FUNCTION_BLOCK FB_MotionInterlocksCommon IMPLEMENTS I_MotionInterlocksCommon
VAR
    {attribute 'hide'}
    iMotionLogger 		: I_MotionLogger;
    {attribute 'hide'}
    bPowerEnabled: BOOL:=FALSE;
   // NC STO Input: TRUE if ok to move
    {attribute 'pytmc' := '
        pv: PLC:bHardwareEnable
        io: i
        field: ZNAM FALSE
        field: ONAM TRUE
        field: DESC TRUE if STO not hit
    '}
    bHardwareEnable AT %I*: BOOL ;

    // Used by the IOC to disable an axis
    {attribute 'pytmc' := '
        pv: PLC:bUserEnable
        io: io
        field: ZNAM DISABLE
        field: ONAM ENABLE
        field: DESC Used to disable power entirely for an axis
    '}
    bUserEnable: BOOL := TRUE;

    {attribute 'hide'}
    bEnable: BOOL;
    {attribute 'hide'}
    bReset : BOOL;
    {attribute 'hide'}
    sMessage : STRING;
    {attribute 'hide'}
    bError : BOOL;
    {attribute 'hide'}
    nErrorID : UDINT;
    {attribute 'hide'}
    bMoveOk : BOOL;
END_VAR

IF ( iMotionLogger = 0) THEN
    // throw an exception
    RETURN;
END_IF

bPowerEnabled := bEnable AND bHardwareEnable;
bPowerEnabled R= NOT bUserEnable;

(*test additional pre-move conditions here*)
bMoveOk := bUserEnable AND bHardwareEnable;

IF NOT bUserEnable OR NOT bHardwareEnable THEN
    bError := TRUE;
    nErrorID:= 11;
    bMoveOk := FALSE;
    IF NOT bUserEnable THEN
        sMessage := 'User enable interlock triggered!';
    ELSE
        sMessage := 'Hardware enbale interlocks triggered!';
    END_IF
END_IF

METHOD PUBLIC CallAfterInit
VAR_INPUT
    iMotionLogger : I_MotionLogger;
END_VAR
THIS^.iMotionLogger := iMotionLogger;
END_METHOD

METHOD DriveCommands
VAR_INPUT
    Enable: BOOL;
    NewMoveReq : BOOL;
END_VAR
THIS^.bEnable := Enable;
THIS^.bPowerEnabled := bEnable AND bHardwareEnable;
END_METHOD

{attribute 'monitoring' := 'variable'}
PROPERTY Error : BOOL
GET
Error := bError;
END_GET
END_PROPERTY

PROPERTY ErrorID : UDINT
GET
ErrorID := nErrorID;
END_GET
END_PROPERTY

//FB_Init is always available implicitly and it is used primarily for initialization.
//The return value is not evaluated. For a specific influence, you can also declare the
//methods explicitly and provide additional code there with the standard initialization
//code. You can evaluate the return value.
METHOD FB_Init: BOOL
VAR_INPUT
    bInitRetains: BOOL; // TRUE: the retain variables are initialized (reset warm / reset cold)
    bInCopyCode: BOOL;  // TRUE: the instance will be copied to the copy code afterward (online change)

    iMotionLogger 		: I_MotionLogger;
END_VAR
THIS^.iMotionLogger := iMotionLogger;
END_METHOD

PROPERTY HardwareEnable : BOOL
GET
END_GET
SET
bHardwareEnable := HardwareEnable;
END_SET
END_PROPERTY

PROPERTY Message : T_MAXSTRING
GET
Message := sMessage;
END_GET
END_PROPERTY

{attribute 'monitoring' := 'variable'}
PROPERTY MoveOk : BOOL
GET
MoveOk := bMoveOk;
END_GET
END_PROPERTY

{attribute 'monitoring' := 'variable'}
PROPERTY PowerEnabled : BOOL
GET
PowerEnabled :=bPowerEnabled;
END_GET
END_PROPERTY

METHOD Reset
THIS^.bError := FALSE;
THIS^.nErrorID:= 0;
THIS^.sMessage:='';
END_METHOD

PROPERTY UserEnable : BOOL
SET
bUserEnable := UserEnable;
END_SET
END_PROPERTY

END_FUNCTION_BLOCK

(* stored: Version 1.1.0.1
   POU FB_MotionInterlocksCommon: Id {b69073ed-2a55-41fc-84a9-b8fe79332e5e}, SpecialFunc None
   Method CallAfterInit: Id {bb25ce30-2def-4497-bead-4e7295fc730f}
   Method DriveCommands: Id {6d01eab2-7989-4c7e-b542-03db7614d447}
   Property Error: Id {21f5c9dd-d9f9-4fb7-a70a-688ad37ac74c}
   Get Get: Id {021721b1-8d55-49d6-a8cf-4547c5e3bcd2}
   Property ErrorID: Id {c58250f8-ae5a-4056-a2ed-503e8b03cb8d}
   Get Get: Id {a1817a62-dd31-4d18-8907-b880a900e971}
   Method FB_Init: Id {ee1048d7-3a0b-4701-a887-c2bc01c18e00}
   Property HardwareEnable: Id {d61e5b05-94b6-4b80-bfd7-0d1f07731219}
   Get Get: Id {de4ec138-0ec0-4fe4-93ac-6a00a13d21e6}
   Set Set: Id {997b3317-ecd2-4d78-ab35-890e6b79db96}
   Property Message: Id {fff95902-de95-4707-8ab7-164e983a966f}
   Get Get: Id {aa8e66bf-be37-477b-a097-6e499951d5ae}
   Property MoveOk: Id {a6c854ac-10d2-4324-b515-25871c48273c}
   Get Get: Id {c6848f02-95c1-4045-9aa0-95260cab536e}
   Property PowerEnabled: Id {6a435248-a266-41ef-9b9c-8e0bf7663a4b}
   Get Get: Id {c27ac7b3-d93e-4dca-97d4-f9f71a18aff4}
   Method Reset: Id {705b0120-de09-4ca3-922f-20b5238adb32}
   Property UserEnable: Id {3dd63e54-e47f-4503-9258-eaac8ea1f82e}
   Set Set: Id {1bc1daba-a9ae-4d73-a148-bfc9f891f3f2} *)
